Staubli VAL3: chkQuickStop.pgx

program chkQuickStop()
  local num l_ni
begin
  //
  bDriveQuickStop=false
  for l_ni=0 to nAxesSum-1
    if nDrvState[l_ni]==12
      bQuickStop[l_ni]=true
    else
      bQuickStop[l_ni]=false
    endIf
    bDriveQuickStop=bDriveQuickStop or bQuickStop[l_ni]
  endFor
end
